// TIA Portal V18 export
ORGANIZATION_BLOCK "Main"   // OB1, LAD, ProgramCycle
TITLE = "Main Program Sweep (Cycle)"
{ S7_Optimized_Access := 'TRUE' }
// stored: SetENOAutomatically false
   VAR_INPUT
      Initial_Call : Bool;   // Initial call of this OB
      Remanence : Bool;   // =True, if remanent data are available
   END_VAR
BEGIN

REGION Network 1
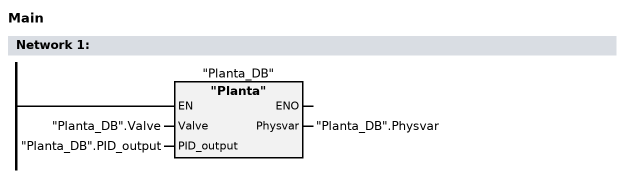
   RUNG wire#powerrail
      "Planta_DB"(Valve := "Planta_DB".Valve, PID_output := "Planta_DB".PID_output, Physvar => "Planta_DB".Physvar)
   END_RUNG
   // the same network as SCL:
   "Planta_DB"(Valve := "Planta_DB".Valve, PID_output := "Planta_DB".PID_output, Physvar => "Planta_DB".Physvar);   // "Planta"
END_REGION
END_ORGANIZATION_BLOCK
